// TIA Portal V19 export
TYPE "LAF_typeDevDiagInstruct"
TITLE = Device Diag Instructions / Device Diag Anweisungen
// This data type contains the structure for the read diagnostic data.  
// 
// **PLC Data types**  
// * [LAF_typeDevDiagModStateMode](../Library%20Types/LAF_typeDevDiagModStateMode.htm)  
// * [LAF_typeDevDiagStructGetDiag](../Library%20Types/LAF_typeDevDiagStructGetDiag.htm)
// Struktur Device Diag Anweisungen
// stored: Access Published
   STRUCT
      log2GeoLaddr { ExternalAccessible := 'False'; ExternalVisible := 'False'; ExternalWritable := 'False'} : HW_IOSYSTEM;   // LOG2GEO address / LOG2GEO Adresse
      log2GeoRetVal { ExternalAccessible := 'False'; ExternalVisible := 'False'; ExternalWritable := 'False'} : Int;   // RetVal instruction / RetVal Anweisung
      log2Geo { ExternalAccessible := 'False'; ExternalVisible := 'False'; ExternalWritable := 'False'} : GEOADDR;   // Geologische Adresse / Geological address
      devStateMode1 { ExternalAccessible := 'False'; ExternalVisible := 'False'; ExternalWritable := 'False'} : "LAF_typeDevDiagStatesMode";   // Konfiguriert / Configured
      devStateMode2 { ExternalAccessible := 'False'; ExternalVisible := 'False'; ExternalWritable := 'False'} : "LAF_typeDevDiagStatesMode";   // Gestoert / Faulty
      devStateMode3 { ExternalAccessible := 'False'; ExternalVisible := 'False'; ExternalWritable := 'False'} : "LAF_typeDevDiagStatesMode";   // Deaktiviert / Deactivated
      devStateMode4 { ExternalAccessible := 'False'; ExternalVisible := 'False'; ExternalWritable := 'False'} : "LAF_typeDevDiagStatesMode";   // Vorhanden / Present
      devStateMode5 { ExternalAccessible := 'False'; ExternalVisible := 'False'; ExternalWritable := 'False'} : "LAF_typeDevDiagStatesMode";   // Problem
      geo2LogLaddr { ExternalAccessible := 'False'; ExternalVisible := 'False'; ExternalWritable := 'False'} : HW_ANY;   // GEO2LOG address / GEO2LOG Adresse
      geo2LogRetVal { ExternalAccessible := 'False'; ExternalVisible := 'False'; ExternalWritable := 'False'} : Int;   // RetVal instruction / RetVal Anweisung
      geo2Log { ExternalAccessible := 'False'; ExternalVisible := 'False'; ExternalWritable := 'False'} : GEOADDR;   // Geologische Adresse / Geological address
      moduleStateMode2 { ExternalAccessible := 'False'; ExternalVisible := 'False'; ExternalWritable := 'False'} : "LAF_typeDevDiagModStateMode";   // Mode 1: konfiguriert, 2: gestoert, 3: deaktiviert, 4: vorhanden, 5: Problem / Mode 1: Configured 2: Faulty 3: Deactivated 4: Present 5: Problem
      moduleStateMode5 { ExternalAccessible := 'False'; ExternalVisible := 'False'; ExternalWritable := 'False'} : "LAF_typeDevDiagModStateMode";   // Mode 1: konfiguriert, 2: gestoert, 3: deaktiviert, 4: vorhanden, 5: Problem / Mode 1: Configured 2: Faulty 3: Deactivated 4: Present 5: Problem
      getDiag { ExternalAccessible := 'False'; ExternalVisible := 'False'; ExternalWritable := 'False'} : "LAF_typeDevDiagStructGetDiag";   // Read diagnostc informationen of a hardware component / Diagnoseinformationen einer Hardware Komponente auslesen
   END_STRUCT;
END_TYPE
